Staubli VAL3: goRemote.pgx

program goRemote()
begin
  call setSpeed()
  movel(pGoRemoteTarget, tTool, mNomSpeed)
  waitEndMove()
end
